/// configuration data that is used during boot to configure the Units equipment
TYPE HandlingDataConfig :
STRUCT
  Simulated : BOOL;
END_STRUCT
END_TYPE

(* stored: Version 1.1.0.1
   DUT HandlingDataConfig: Id {5c208c65-6e03-42ce-b87e-19afbbb4d0a1} *)
